// TIA Portal V20 export
DATA_BLOCK "HmiInterface"   // DB97
// stored: Access Published, MemoryReserve 100, Namespace Unit1.Em6
   VAR
      em : "LAF_typeEmInterface";
      emHomedCheck : "Unit1.Em6.typeEmHomedCheck";
      cm : "Unit1.Em6.typeCmInterface";
      visionUnit : "LER_typeSequenceInterface";
      visionController : "LER_typeSequenceInterface";
      qrRead : "LER_typeSequenceInterface";
   END_VAR
   VAR RETAIN
      cmVisionUnitAxisZ : "LBC_typeAxis64PosInterface";
      cmVisionPusherSupportUpDown : "LBC_typeTwoWayActuatorInterface";
      cmVisionTriggerSensor : "LBC_typeDigitalSignalInterface";
      cmVisionController : "LER_typeVisionInterface";
      cmQrReader : "LER_typeSRX300Interface";
      cmQrReadHandy : "LER_typeDM8700Interface";
      cmVisionUnitAxisZ_TorqueCal : "LER_typeServoTorqueCalInterface";
      cmVisionDataConvert : "LER_typeVisionResultData";
      GaugeRnRType1 : "LER_typeCount";
      GaugeRnRType3 : "LER_typeCount";
      GaugeRnRType3Parts : "LER_typeCount";
      visionTriggerSensorNotDetectedCount : "LER_typeAlarmCounterInterface";
      cmVisionHistory : "LER_typeVisionHistory";
      cmVisionQrHistory : "LER_typeQrHistory";
   END_VAR
BEGIN
END_DATA_BLOCK
